// TIA Portal project "test" (V15)

(* hardware
DEVICE "S7-1200 station_1"  S7-1200 Station
   slot 0: "Rack_0"  S7-1200 Rack  Rack  V1.0
   slot 1: "PLC_1"  CPU 1214C DC/DC/Rly  6ES7 214-1HG40-0XB0  V4.2
*)

// ===== PLC "PLC_1"  CPU 1214C DC/DC/Rly =====

VAR_GLOBAL   // PLC tag table "Default tag table"
   "X" AT %I0.0 : Bool;   // Cảm biến phát hiện vật vào đúng vị trí
   "a1" AT %I0.1 : Bool;   // Cảm biến hành trình van A đã kẹp vật
   "b0" AT %I0.2 : Bool;   // Cảm biến hành trình B đã thu về
   "b1" AT %I0.3 : Bool;   // Xy lanh B đã đi ra
   "c0" AT %I0.4 : Bool;   // Xy lanh C thu về
   "c1" AT %I0.5 : Bool;   // Xy lanh C đi ra
   "A+" AT %Q0.0 : Bool;   // Van A đi ra
   "B-" AT %Q0.1 : Bool;   // Van B thu về
   "B+" AT %Q0.2 : Bool;   // Van B đi ra
   "C-" AT %Q0.3 : Bool;   // Van C thu về
   "C+" AT %Q0.4 : Bool;   // Van C đi ra
   "START" AT %M0.0 : Bool;
   "STOP" AT %M0.1 : Bool;   // THỰC HIỆN XONG CHU TRÌNH THÌ DỪNG
   "EM-STOP" AT %M0.2 : Bool;   // DỪNG TẠI THỜI ĐIỂM BẤT KỲ, KHI KHẮC PHỤC XONG CHẠY TIẾP TỪ VỊ TRÍ DỪNG
   "MANUAL" AT %M0.3 : Bool;
   "AUTO" AT %M0.4 : Bool;
   "Tag_1" AT %M1.0 : Bool;
   "Tag_2" AT %M1.1 : Bool;
   "Tag_3" AT %M1.2 : Bool;
   "Tag_4" AT %M1.3 : Bool;
   "Tag_5" AT %M1.4 : Bool;
   "Tag_6" AT %M1.5 : Bool;
   "BT-Control" AT %Q0.5 : Bool;   // Băng tải chạy
   "S0" AT %M5.0 : Bool;   // BĂNG TẢI CHẠY
   "S1" AT %M5.1 : Bool;   // XY LANH A KẸP VẬT
   "S2" AT %M5.2 : Bool;   // XY LANH B DI CHUYỂN ĐỂ UỐN VẬT
   "S3" AT %M5.3 : Bool;   // XY LANH B THU VỀ
   "S4" AT %M5.4 : Bool;   // XY LANH C CHUYỂN SANG TRÁI UỐN VẬT
   "S5" AT %M5.5 : Bool;   // XY LANH C THU VỀ
   "S6" AT %M5.6 : Bool;   // XY LANH A THU VỀ
   "a0" AT %I0.6 : Bool;   // Cảm biến A thu về
END_VAR

FUNCTION "HAND" : Void   // FC1, LAD
{ S7_Optimized_Access := 'TRUE' }
VERSION : 0.1
BEGIN

REGION Network 1: Van A đi ra
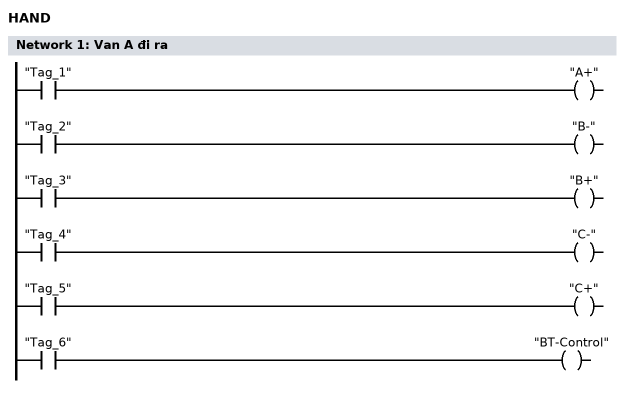
   RUNG wire#powerrail
      Contact( "Tag_1" )
      Coil( "A+" )
   END_RUNG
   RUNG wire#powerrail
      Contact( "Tag_2" )
      Coil( "B-" )
   END_RUNG
   RUNG wire#powerrail
      Contact( "Tag_3" )
      Coil( "B+" )
   END_RUNG
   RUNG wire#powerrail
      Contact( "Tag_4" )
      Coil( "C-" )
   END_RUNG
   RUNG wire#powerrail
      Contact( "Tag_5" )
      Coil( "C+" )
   END_RUNG
   RUNG wire#powerrail
      Contact( "Tag_6" )
      Coil( "BT-Control" )
   END_RUNG
   // the same network as SCL:
   "A+" := "Tag_1";
   "B-" := "Tag_2";
   "B+" := "Tag_3";
   "C-" := "Tag_4";
   "C+" := "Tag_5";
   "BT-Control" := "Tag_6";
END_REGION
END_FUNCTION

FUNCTION "AUTO-PRO" : Void   // FC2, LAD
{ S7_Optimized_Access := 'TRUE' }
VERSION : 0.1
BEGIN

REGION Network 1: BĂNG TẢI CHẠY
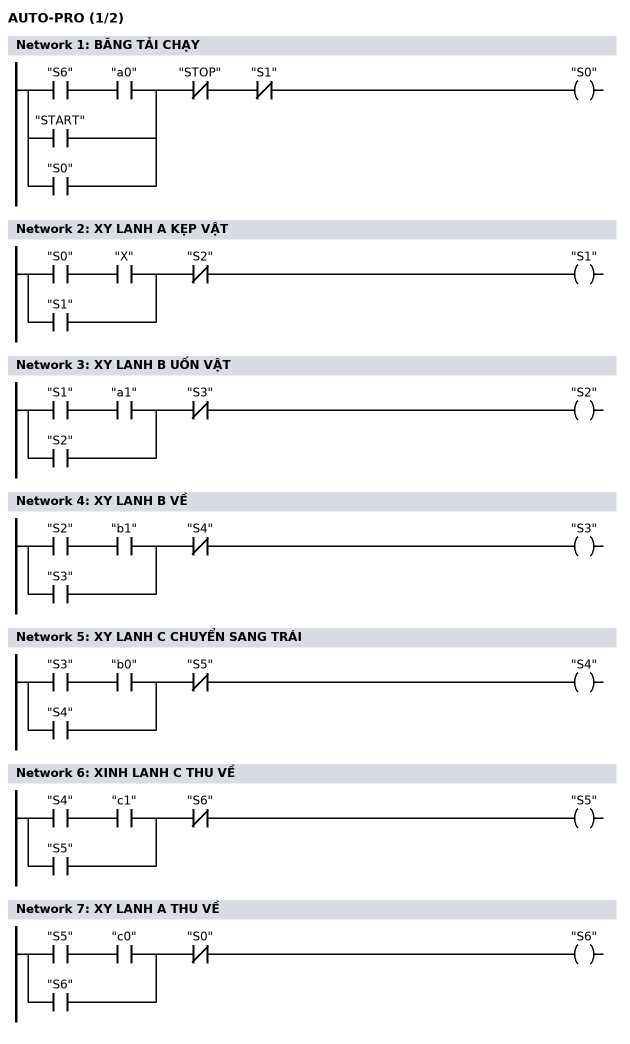
   RUNG wire#powerrail
      Contact( "S6" )
      Contact( "a0" )
      wire#w1
      I_Contact( "STOP" )
      I_Contact( "S1" )
      Coil( "S0" )
   END_RUNG
   RUNG wire#powerrail
      Contact( "START" )
   END_RUNG wire#w1
   RUNG wire#powerrail
      Contact( "S0" )
   END_RUNG wire#w1
   // the same network as SCL:
   "S0" := (("S6" AND "a0") OR "START" OR "S0") AND NOT "STOP" AND NOT "S1";
END_REGION

REGION Network 2: XY LANH A KẸP VẬT
   RUNG wire#powerrail
      Contact( "S0" )
      Contact( "X" )
      wire#w1
      I_Contact( "S2" )
      Coil( "S1" )
   END_RUNG
   RUNG wire#powerrail
      Contact( "S1" )
   END_RUNG wire#w1
   // the same network as SCL:
   "S1" := (("S0" AND "X") OR "S1") AND NOT "S2";
END_REGION

REGION Network 3: XY LANH B UỐN VẬT
   RUNG wire#powerrail
      Contact( "S1" )
      Contact( "a1" )
      wire#w1
      I_Contact( "S3" )
      Coil( "S2" )
   END_RUNG
   RUNG wire#powerrail
      Contact( "S2" )
   END_RUNG wire#w1
   // the same network as SCL:
   "S2" := (("S1" AND "a1") OR "S2") AND NOT "S3";
END_REGION

REGION Network 4: XY LANH B VỀ
   RUNG wire#powerrail
      Contact( "S2" )
      Contact( "b1" )
      wire#w1
      I_Contact( "S4" )
      Coil( "S3" )
   END_RUNG
   RUNG wire#powerrail
      Contact( "S3" )
   END_RUNG wire#w1
   // the same network as SCL:
   "S3" := (("S2" AND "b1") OR "S3") AND NOT "S4";
END_REGION

REGION Network 5: XY LANH C CHUYỂN SANG TRÁI
   RUNG wire#powerrail
      Contact( "S3" )
      Contact( "b0" )
      wire#w1
      I_Contact( "S5" )
      Coil( "S4" )
   END_RUNG
   RUNG wire#powerrail
      Contact( "S4" )
   END_RUNG wire#w1
   // the same network as SCL:
   "S4" := (("S3" AND "b0") OR "S4") AND NOT "S5";
END_REGION

REGION Network 6: XINH LANH C THU VỀ
   RUNG wire#powerrail
      Contact( "S4" )
      Contact( "c1" )
      wire#w1
      I_Contact( "S6" )
      Coil( "S5" )
   END_RUNG
   RUNG wire#powerrail
      Contact( "S5" )
   END_RUNG wire#w1
   // the same network as SCL:
   "S5" := (("S4" AND "c1") OR "S5") AND NOT "S6";
END_REGION

REGION Network 7: XY LANH A THU VỀ
   RUNG wire#powerrail
      Contact( "S5" )
      Contact( "c0" )
      wire#w1
      I_Contact( "S0" )
      Coil( "S6" )
   END_RUNG
   RUNG wire#powerrail
      Contact( "S6" )
   END_RUNG wire#w1
   // the same network as SCL:
   "S6" := (("S5" AND "c0") OR "S6") AND NOT "S0";
END_REGION

REGION Network 8: Băng tải chạy
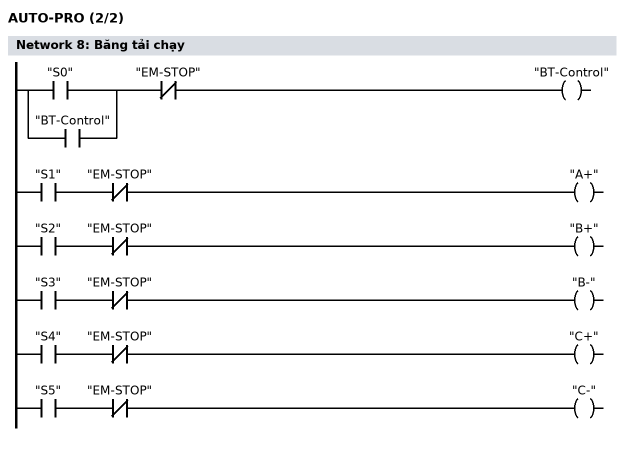
   RUNG wire#powerrail
      Contact( "S0" )
      wire#w1
      I_Contact( "EM-STOP" )
      Coil( "BT-Control" )
   END_RUNG
   RUNG wire#powerrail
      Contact( "BT-Control" )
   END_RUNG wire#w1
   RUNG wire#powerrail
      Contact( "S1" )
      I_Contact( "EM-STOP" )
      Coil( "A+" )
   END_RUNG
   RUNG wire#powerrail
      Contact( "S2" )
      I_Contact( "EM-STOP" )
      Coil( "B+" )
   END_RUNG
   RUNG wire#powerrail
      Contact( "S3" )
      I_Contact( "EM-STOP" )
      Coil( "B-" )
   END_RUNG
   RUNG wire#powerrail
      Contact( "S4" )
      I_Contact( "EM-STOP" )
      Coil( "C+" )
   END_RUNG
   RUNG wire#powerrail
      Contact( "S5" )
      I_Contact( "EM-STOP" )
      Coil( "C-" )
   END_RUNG
   // the same network as SCL:
   "BT-Control" := ("S0" OR "BT-Control") AND NOT "EM-STOP";
   "A+" := "S1" AND NOT "EM-STOP";
   "B+" := "S2" AND NOT "EM-STOP";
   "B-" := "S3" AND NOT "EM-STOP";
   "C+" := "S4" AND NOT "EM-STOP";
   "C-" := "S5" AND NOT "EM-STOP";
END_REGION
END_FUNCTION

ORGANIZATION_BLOCK "Main"   // OB1, LAD, ProgramCycle
TITLE = "Main Program Sweep (Cycle)"
{ S7_Optimized_Access := 'TRUE' }
VERSION : 0.1
   VAR_INPUT
      Initial_Call : Bool;   // Initial call of this OB
      Remanence : Bool;   // =True, if remanent data are available
   END_VAR
BEGIN

REGION Network 1
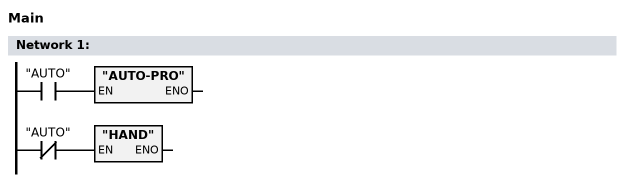
   RUNG wire#powerrail
      Contact( "AUTO" )
      "AUTO-PRO"()
   END_RUNG
   RUNG wire#powerrail
      I_Contact( "AUTO" )
      "HAND"()
   END_RUNG
   // the same network as SCL:
   IF "AUTO" THEN "AUTO-PRO"(); END_IF;
   IF NOT "AUTO" THEN "HAND"(); END_IF;
END_REGION
END_ORGANIZATION_BLOCK